// TIA Portal V20 export
DATA_BLOCK "ET500SP_503"   // DB249
// stored: MemoryReserve 100
   VAR
      "SP503.00 LEFT UNWINDER RADIUS MEASURE" : LReal;
      "SP503.01 RIGHT UNWINDER RADIUS MEASURE" : LReal;
      "SP503.02 UNWINDER LOADCELL" : LReal;
      "SP503.03 CUTTER EPC SENSOR" : LReal;
   END_VAR
BEGIN
END_DATA_BLOCK
